// TIA Portal V16 export
// export: Created 2021-10-20T13:41:55.0672226Z, ExportSetting WithDefaults, DisplayName Totally Integrated Automation Portal, DisplayVersion V16, DisplayName TIA Portal Version Control Interface, DisplayVersion V16, DisplayName TIA Portal Openness, DisplayVersion V16, DisplayName TIA Portal Teamcenter Gateway, DisplayVersion V16, DisplayName SINAMICS Startdrive Advanced, DisplayVersion V16, DisplayName SINAMICS Startdrive G130, G150, S120, S150, SINAMICS MV, S210, DisplayVersion V16, DisplayName SINAMICS Startdrive G110M, G120, G120C, G120D, G120P, DisplayVersion V16, DisplayName STEP 7 Professional, DisplayVersion V16, DisplayName STEP 7 Safety, DisplayVersion V16, DisplayName WinCC Advanced, DisplayVersion V16
ORGANIZATION_BLOCK "Cyclic interrupt"   // OB30, LAD, CyclicInterrupt
TITLE = HMI Data Exchange
{ S7_Optimized_Access := 'TRUE' }
VERSION : 0.1
// This block controls the data exchange between this PLC (A2L) and the Indoor Room PLC's for Rooms 4 & 5.
// stored: AutoNumber true, IsIECCheckEnabled false, SetENOAutomatically false
   VAR_INPUT
      Initial_Call : Bool;   // Initial call of this OB
      Event_Count : Int;   // Events discarded
   END_VAR
BEGIN

REGION Network 1: Rm4 ID North DB Moves
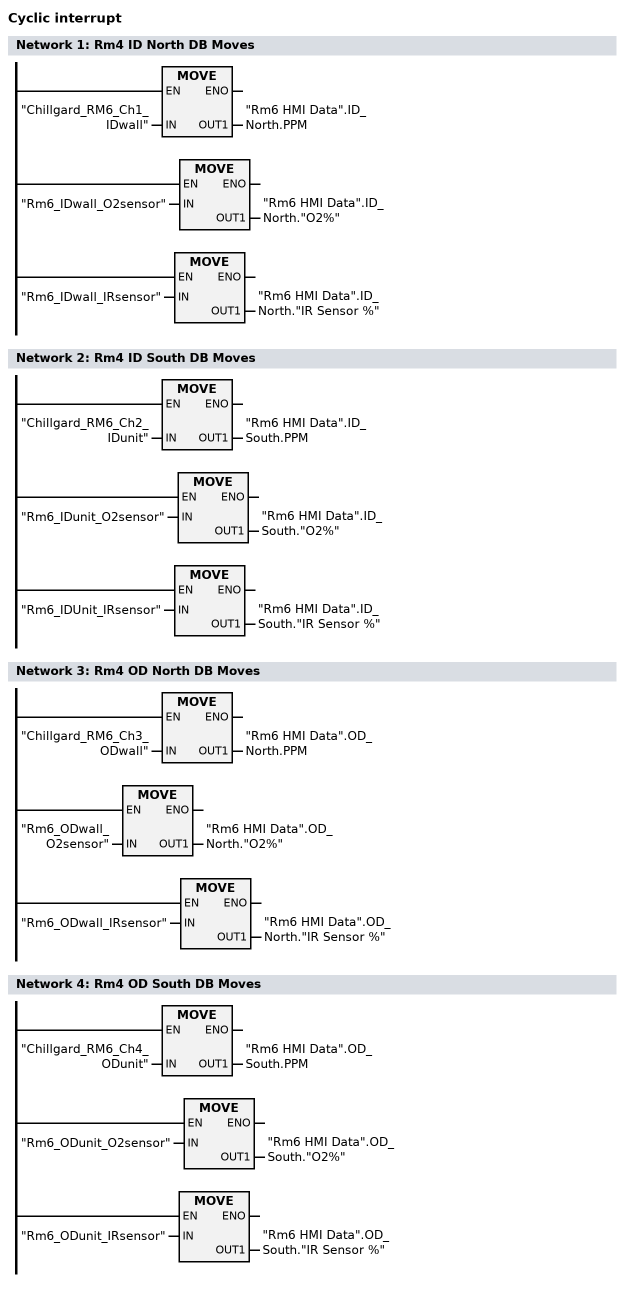
   RUNG wire#powerrail
      Move(in := "Chillgard_RM6_Ch1_IDwall", out1 => "Rm6 HMI Data".ID_North.PPM)
   END_RUNG
   RUNG wire#powerrail
      Move(in := "Rm6_IDwall_O2sensor", out1 => "Rm6 HMI Data".ID_North."O2%")
   END_RUNG
   RUNG wire#powerrail
      Move(in := "Rm6_IDwall_IRsensor", out1 => "Rm6 HMI Data".ID_North."IR Sensor %")
   END_RUNG
   // the same network as SCL:
   "Rm6 HMI Data".ID_North.PPM := "Chillgard_RM6_Ch1_IDwall";
   "Rm6 HMI Data".ID_North."O2%" := "Rm6_IDwall_O2sensor";
   "Rm6 HMI Data".ID_North."IR Sensor %" := "Rm6_IDwall_IRsensor";
END_REGION

REGION Network 2: Rm4 ID South DB Moves
   RUNG wire#powerrail
      Move(in := "Chillgard_RM6_Ch2_IDunit", out1 => "Rm6 HMI Data".ID_South.PPM)
   END_RUNG
   RUNG wire#powerrail
      Move(in := "Rm6_IDunit_O2sensor", out1 => "Rm6 HMI Data".ID_South."O2%")
   END_RUNG
   RUNG wire#powerrail
      Move(in := "Rm6_IDUnit_IRsensor", out1 => "Rm6 HMI Data".ID_South."IR Sensor %")
   END_RUNG
   // the same network as SCL:
   "Rm6 HMI Data".ID_South.PPM := "Chillgard_RM6_Ch2_IDunit";
   "Rm6 HMI Data".ID_South."O2%" := "Rm6_IDunit_O2sensor";
   "Rm6 HMI Data".ID_South."IR Sensor %" := "Rm6_IDUnit_IRsensor";
END_REGION

REGION Network 3: Rm4 OD North DB Moves
   RUNG wire#powerrail
      Move(in := "Chillgard_RM6_Ch3_ODwall", out1 => "Rm6 HMI Data".OD_North.PPM)
   END_RUNG
   RUNG wire#powerrail
      Move(in := "Rm6_ODwall_O2sensor", out1 => "Rm6 HMI Data".OD_North."O2%")
   END_RUNG
   RUNG wire#powerrail
      Move(in := "Rm6_ODwall_IRsensor", out1 => "Rm6 HMI Data".OD_North."IR Sensor %")
   END_RUNG
   // the same network as SCL:
   "Rm6 HMI Data".OD_North.PPM := "Chillgard_RM6_Ch3_ODwall";
   "Rm6 HMI Data".OD_North."O2%" := "Rm6_ODwall_O2sensor";
   "Rm6 HMI Data".OD_North."IR Sensor %" := "Rm6_ODwall_IRsensor";
END_REGION

REGION Network 4: Rm4 OD South DB Moves
   RUNG wire#powerrail
      Move(in := "Chillgard_RM6_Ch4_ODunit", out1 => "Rm6 HMI Data".OD_South.PPM)
   END_RUNG
   RUNG wire#powerrail
      Move(in := "Rm6_ODunit_O2sensor", out1 => "Rm6 HMI Data".OD_South."O2%")
   END_RUNG
   RUNG wire#powerrail
      Move(in := "Rm6_ODunit_IRsensor", out1 => "Rm6 HMI Data".OD_South."IR Sensor %")
   END_RUNG
   // the same network as SCL:
   "Rm6 HMI Data".OD_South.PPM := "Chillgard_RM6_Ch4_ODunit";
   "Rm6 HMI Data".OD_South."O2%" := "Rm6_ODunit_O2sensor";
   "Rm6 HMI Data".OD_South."IR Sensor %" := "Rm6_ODunit_IRsensor";
END_REGION
END_ORGANIZATION_BLOCK
